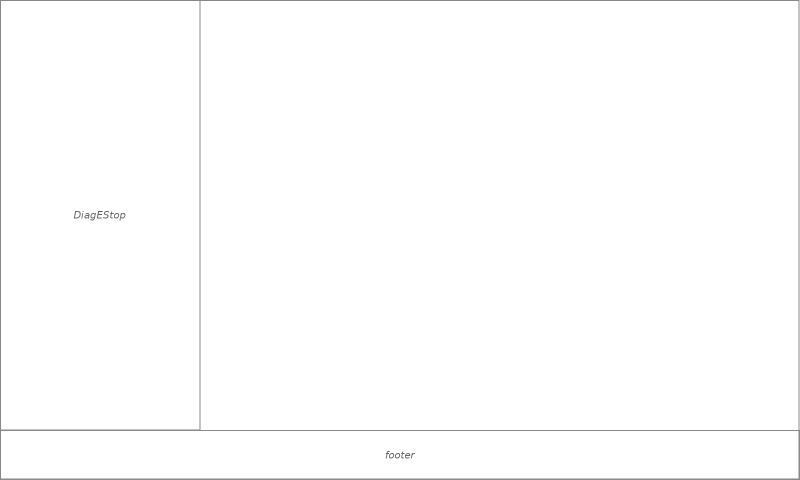
VISUALIZATION FB_Diag  // 800x480
    Frame (0,430 800x50)
        shows footer()
    Frame (0,0 200x430)
        shows DiagEStop(state := safetyDiag.sEStopState, bits := safetyDiag.eStopDiagBits, blockName := 'Emergência')
END_VISUALIZATION

(* stored: Version 1.1.0.1, ProductVersion 3.1.4024.12
   Visu FB_Diag: Id {3ede58e4-3d1c-41e7-b269-dc91fc2d33ee} *)
